DATA_BLOCK "DATA_CONFIG"
{ DB_Accessible_From_OPC_UA := 'FALSE' ;
 S7_Optimized_Access := 'TRUE' }
VERSION : 0.1
NON_RETAIN
   VAR
      PLCVersion { ExternalWritable := 'False'} : String["DIM_STRINGNAME"];   // scritto su Settings
      PLCVersion1 : Int;
      PLCVersion2 : Int;
      PLCVersion3 : Int;
      PLCVersion4 : Int;
      CFGVersion : Int;   // PLCVersion1 * 100 + PLCVersion2
      SerType : Int;   // tipo dati Deserialize
      SerCurrInd : Int;   // indice blocco corrente Deserialize
      SerCurrLast : Int;   // indice ultimo blocco Deserialize
      SerIndStat : Int;
      SerTotRot : Real;
      ConfigReqTime { ExternalAccessible := 'False'; ExternalVisible := 'False'; ExternalWritable := 'False'} : Time;   // NON USATO
      ConfigReqTimeout { ExternalAccessible := 'False'; ExternalVisible := 'False'; ExternalWritable := 'False'} : ULInt;   // NON USATO
      ConfigAckTime { ExternalAccessible := 'False'; ExternalVisible := 'False'; ExternalWritable := 'False'} : Time;   // NON USATO
      ConfigAckTimeout { ExternalAccessible := 'False'; ExternalVisible := 'False'; ExternalWritable := 'False'} : ULInt;   // NON USATO
      ConfigSaveReqTime : Time;
      ConfigSaveReqTimeout : ULInt;
      ConfigSaveReqStart : Bool;
      TabstatReqTime : Time;
      TabstatReqTimeout : ULInt;
      ProgReqHMITime : Time;
      ProgReqHMITimeout : ULInt;
      SaveConfigReq { ExternalAccessible := 'False'; ExternalVisible := 'False'; ExternalWritable := 'False'} : Bool;
      SaveConfigCurrStep { ExternalAccessible := 'False'; ExternalVisible := 'False'; ExternalWritable := 'False'} : Int;
      DeletingFile { ExternalAccessible := 'False'; ExternalVisible := 'False'; ExternalWritable := 'False'} : Bool;
      SavingFile : Bool;   // Scrittura file su WebServer in corso
      DebugInd { ExternalAccessible := 'False'; ExternalVisible := 'False'; ExternalWritable := 'False'} : Int;
      DebugInd2 { ExternalAccessible := 'False'; ExternalVisible := 'False'; ExternalWritable := 'False'} : Int;
      Config_Header { ExternalWritable := 'False'} : Array[0.."MAX_HEADER"] of Int;   // SN,FileType,FileTypeVersion,FileVersion
      AxisFunInd : Array[0.."MAX_ASSEFUNIND"] of Int;
      InInd : Array[0.."MAX_STATOBOOL"] of Int;
      OutInd : Array[0.."MAX_STATOBOOL"] of Int;
      ParamString : Array[0.."MAX_PARAMSTRING"] of String["DIM_STRINGNAME"];
      ParamBool : Array[0.."MAX_PARAMBOOL"] of Bool;
      ParamInt : Array[0.."MAX_PARAMINT"] of Int;
      ParamRealCfg : Array[0.."MAX_PARAMREAL"] of Real;
      ParamReal : Array[0.."MAX_PARAMREAL"] of Real;
      ParamRealType : Array[0.."MAX_PARAMREAL"] of Int;
      ParamRealFC { ExternalAccessible := 'False'; ExternalVisible := 'False'; ExternalWritable := 'False'} : Array[0.."MAX_PARAMREAL"] of Real;
      ParamRealOffset : Array[0.."MAX_PARAMREAL"] of Real;
      IO_Name : Array[0.."MAX_IO"] of String["DIM_STRINGNAME"];
      IO_Param { S7_SetPoint := 'False'} : Array[0.."MAX_IO"] of "Type_IOParam";
      Axis_Name : Array[0.."MAX_ASSE"] of String["DIM_STRINGID"];
      Axis_Param { S7_SetPoint := 'False'} : Array[0.."MAX_ASSE"] of "Type_AxisParam";
      Axis { S7_SetPoint := 'False'} : Array[0.."MAX_ASSE"] of "Type_Axis";
      Input { S7_SetPoint := 'False'} : Array[0.."MAX_INPUT"] of "Type_Input";
      Input_Param { S7_SetPoint := 'False'} : Array[0.."MAX_INPUT"] of "Type_InputParam";
      Feedback { S7_SetPoint := 'False'} : Array[0.."MAX_FEEDBACK"] of "Type_Feedback";
      Feedback_Param { S7_SetPoint := 'False'} : Array[0.."MAX_FEEDBACK"] of "Type_FeedbackParam";
      PID { ExternalAccessible := 'False'; ExternalVisible := 'False'; ExternalWritable := 'False'; S7_SetPoint := 'False'} : Array[0.."MAX_PID"] of "Type_PID";
      PID_Param { S7_SetPoint := 'False'} : Array[0.."MAX_PID"] of "Type_PIDParam";
      Output { S7_SetPoint := 'False'} : Array[0.."MAX_OUTPUT"] of "Type_Output";
      Output_Param { S7_SetPoint := 'False'} : Array[0.."MAX_OUTPUT"] of "Type_OutputParam";
      Motor { S7_SetPoint := 'False'} : Array[0.."MAX_MOTORE"] of "Type_Motor";
      Motor_Config : Array[0.."MAX_MOTORE"] of Bool;
      Motor_Selectable : Array[0.."MAX_MOTORE"] of Bool;
      Motor_LSInd : Array[0.."MAX_MOTORE"] of Int;
      Motor_LS2Ind : Array[0.."MAX_MOTORE"] of Int;
      Motor_CmdInd : Array[0.."MAX_MOTORE"] of Int;
      Motor_Cmd1Ind : Array[0.."MAX_MOTORE"] of Int;
      Motor_Cmd2Ind : Array[0.."MAX_MOTORE"] of Int;
      Motor_Cmd3Ind : Array[0.."MAX_MOTORE"] of Int;
      Motor_StatInd : Array[0.."MAX_MOTORE"] of Int;
      Motor_TRInd : Array[0.."MAX_MOTORE"] of Int;
      Motor_TR2Ind : Array[0.."MAX_MOTORE"] of Int;
      Motor_StartingInd : Array[0.."MAX_MOTORE"] of Int;
      Alarm_Name : Array[0.."MAX_ALARM"] of String["DIM_STRINGNAME"];
      Alarm_Param { S7_SetPoint := 'False'} : Array[0.."MAX_ALARM"] of "Type_AlarmParam";
      Stop_Num : Int;
      Stop_Name : Array[0.."MAX_STOP"] of String["DIM_STRINGNAME"];
      Stop_Ind : Array[0.."MAX_STOP"] of Int;
      Maint_Name : Array[0.."MAX_MAINT"] of String["DIM_STRINGNAME"];
      Maint_Param { S7_SetPoint := 'False'} : Array[0.."MAX_MAINT"] of "Type_MaintParam";
      Toolset_Name { S7_SetPoint := 'True'} : Array[0.."MAX_TOOLSET"] of String["DIM_STRINGNAME"];
      Toolset_Param { S7_SetPoint := 'False'} : Array[0.."MAX_TOOLSET"] of "Type_ToolsetParam";
      UM_FC : Array[0.."MAX_UM"] of Real;
      UM_FC_Met { ExternalAccessible := 'False'; ExternalVisible := 'False'; ExternalWritable := 'False'} : Array[0.."MAX_UM"] of Real;
      UM_FC_Imp { ExternalAccessible := 'False'; ExternalVisible := 'False'; ExternalWritable := 'False'} : Array[0.."MAX_UM"] of Real;
   END_VAR
   VAR RETAIN
      UM_Offset : Array[0.."MAX_UM"] of Real;
   END_VAR
   VAR
      UM_Offset_Met { ExternalAccessible := 'False'; ExternalVisible := 'False'; ExternalWritable := 'False'} : Array[0.."MAX_UM"] of Real;
      UM_Offset_Imp { ExternalAccessible := 'False'; ExternalVisible := 'False'; ExternalWritable := 'False'} : Array[0.."MAX_UM"] of Real;
   END_VAR
   VAR RETAIN
      UM_NDec : Array[0.."MAX_UM"] of Int;
   END_VAR
   VAR
      UM_NDec_Met { ExternalAccessible := 'False'; ExternalVisible := 'False'; ExternalWritable := 'False'} : Array[0.."MAX_UM"] of Int;
      UM_NDec_Imp { ExternalAccessible := 'False'; ExternalVisible := 'False'; ExternalWritable := 'False'} : Array[0.."MAX_UM"] of Int;
   END_VAR
   VAR RETAIN
      UM_Name : Array[0.."MAX_UM"] of String["DIM_STRINGUMNAME"];
   END_VAR
   VAR
      UM_Name_Met { ExternalAccessible := 'False'; ExternalVisible := 'False'; ExternalWritable := 'False'} : Array[0.."MAX_UM"] of String["DIM_STRINGUMNAME"];
      UM_Name_Imp { ExternalAccessible := 'False'; ExternalVisible := 'False'; ExternalWritable := 'False'} : Array[0.."MAX_UM"] of String["DIM_STRINGUMNAME"];
   END_VAR
   VAR RETAIN
      Teach { S7_SetPoint := 'False'} : "Type_Teach";
   END_VAR
   VAR
      Seq { ExternalAccessible := 'False'; ExternalVisible := 'False'; ExternalWritable := 'False'; S7_SetPoint := 'False'} : "Type_Seq";
      HMIAdd0 { ExternalAccessible := 'False'; ExternalVisible := 'False'; ExternalWritable := 'False'} : Int;
   END_VAR


BEGIN
   PLCVersion := '0';
   ConfigReqTime := T#0MS;
   ConfigReqTimeout := 4000;
   ConfigAckTimeout := 4000;
   ConfigSaveReqTimeout := 1500;
   TabstatReqTimeout := 800;
   ProgReqHMITimeout := 1500;
   DebugInd := -1;
   DebugInd2 := -1;
   AxisFunInd[0] := -1;
   AxisFunInd[1] := -1;
   AxisFunInd[2] := -1;
   AxisFunInd[3] := -1;
   AxisFunInd[4] := -1;
   AxisFunInd[5] := -1;
   AxisFunInd[6] := -1;
   AxisFunInd[7] := -1;
   AxisFunInd[8] := -1;
   AxisFunInd[9] := -1;
   AxisFunInd[10] := -1;
   AxisFunInd[11] := -1;
   AxisFunInd[12] := -1;
   AxisFunInd[13] := -1;
   AxisFunInd[14] := -1;
   AxisFunInd[15] := -1;
   AxisFunInd[16] := -1;
   AxisFunInd[17] := -1;
   AxisFunInd[18] := -1;
   AxisFunInd[19] := -1;
   AxisFunInd[20] := -1;
   AxisFunInd[21] := -1;
   AxisFunInd[22] := -1;
   AxisFunInd[23] := -1;
   AxisFunInd[24] := -1;
   AxisFunInd[25] := -1;
   AxisFunInd[26] := -1;
   AxisFunInd[27] := -1;
   AxisFunInd[28] := -1;
   AxisFunInd[29] := -1;
   AxisFunInd[30] := -1;
   AxisFunInd[31] := -1;
   AxisFunInd[32] := -1;
   AxisFunInd[33] := -1;
   AxisFunInd[34] := -1;
   AxisFunInd[35] := -1;
   AxisFunInd[36] := -1;
   AxisFunInd[37] := -1;
   AxisFunInd[38] := -1;
   AxisFunInd[39] := -1;
   AxisFunInd[40] := -1;
   AxisFunInd[41] := -1;
   AxisFunInd[42] := -1;
   AxisFunInd[43] := -1;
   AxisFunInd[44] := -1;
   AxisFunInd[45] := -1;
   AxisFunInd[46] := -1;
   AxisFunInd[47] := -1;
   AxisFunInd[48] := -1;
   AxisFunInd[49] := -1;
   AxisFunInd[50] := -1;
   AxisFunInd[51] := -1;
   AxisFunInd[52] := -1;
   AxisFunInd[53] := -1;
   AxisFunInd[54] := -1;
   AxisFunInd[55] := -1;
   AxisFunInd[56] := -1;
   AxisFunInd[57] := -1;
   AxisFunInd[58] := -1;
   AxisFunInd[59] := -1;
   AxisFunInd[60] := -1;
   AxisFunInd[61] := -1;
   AxisFunInd[62] := -1;
   AxisFunInd[63] := -1;
   AxisFunInd[64] := -1;
   AxisFunInd[65] := -1;
   AxisFunInd[66] := -1;
   AxisFunInd[67] := -1;
   AxisFunInd[68] := -1;
   AxisFunInd[69] := -1;
   AxisFunInd[70] := -1;
   AxisFunInd[71] := -1;
   InInd[0] := -1;
   InInd[1] := -1;
   InInd[2] := -1;
   InInd[3] := -1;
   InInd[4] := -1;
   InInd[5] := -1;
   InInd[6] := -1;
   InInd[7] := -1;
   InInd[8] := -1;
   InInd[9] := -1;
   InInd[10] := -1;
   InInd[11] := -1;
   InInd[12] := -1;
   InInd[13] := -1;
   InInd[14] := -1;
   InInd[15] := -1;
   InInd[16] := -1;
   InInd[17] := -1;
   InInd[18] := -1;
   InInd[19] := -1;
   InInd[20] := -1;
   InInd[21] := -1;
   InInd[22] := -1;
   InInd[23] := -1;
   InInd[24] := -1;
   InInd[25] := -1;
   InInd[26] := -1;
   InInd[27] := -1;
   InInd[28] := -1;
   InInd[29] := -1;
   InInd[30] := -1;
   InInd[31] := -1;
   InInd[32] := -1;
   InInd[33] := -1;
   InInd[34] := -1;
   InInd[35] := -1;
   InInd[36] := -1;
   InInd[37] := -1;
   InInd[38] := -1;
   InInd[39] := -1;
   InInd[40] := -1;
   InInd[41] := -1;
   InInd[42] := -1;
   InInd[43] := -1;
   InInd[44] := -1;
   InInd[45] := -1;
   InInd[46] := -1;
   InInd[47] := -1;
   InInd[48] := -1;
   InInd[49] := -1;
   InInd[50] := -1;
   InInd[51] := -1;
   InInd[52] := -1;
   InInd[53] := -1;
   InInd[54] := -1;
   InInd[55] := -1;
   InInd[56] := -1;
   InInd[57] := -1;
   InInd[58] := -1;
   InInd[59] := -1;
   InInd[60] := -1;
   InInd[61] := -1;
   InInd[62] := -1;
   InInd[63] := -1;
   InInd[64] := -1;
   InInd[65] := -1;
   InInd[66] := -1;
   InInd[67] := -1;
   InInd[68] := -1;
   InInd[69] := -1;
   InInd[70] := -1;
   InInd[71] := -1;
   InInd[72] := -1;
   InInd[73] := -1;
   InInd[74] := -1;
   InInd[75] := -1;
   InInd[76] := -1;
   InInd[77] := -1;
   InInd[78] := -1;
   InInd[79] := -1;
   InInd[80] := -1;
   InInd[81] := -1;
   InInd[82] := -1;
   InInd[83] := -1;
   InInd[84] := -1;
   InInd[85] := -1;
   InInd[86] := -1;
   InInd[87] := -1;
   InInd[88] := -1;
   InInd[89] := -1;
   InInd[90] := -1;
   InInd[91] := -1;
   InInd[92] := -1;
   InInd[93] := -1;
   InInd[94] := -1;
   InInd[95] := -1;
   InInd[96] := -1;
   InInd[97] := -1;
   InInd[98] := -1;
   InInd[99] := -1;
   InInd[100] := -1;
   InInd[101] := -1;
   InInd[102] := -1;
   InInd[103] := -1;
   InInd[104] := -1;
   InInd[105] := -1;
   InInd[106] := -1;
   InInd[107] := -1;
   InInd[108] := -1;
   InInd[109] := -1;
   InInd[110] := -1;
   InInd[111] := -1;
   InInd[112] := -1;
   InInd[113] := -1;
   InInd[114] := -1;
   InInd[115] := -1;
   InInd[116] := -1;
   InInd[117] := -1;
   InInd[118] := -1;
   InInd[119] := -1;
   InInd[120] := -1;
   InInd[121] := -1;
   InInd[122] := -1;
   InInd[123] := -1;
   InInd[124] := -1;
   InInd[125] := -1;
   InInd[126] := -1;
   InInd[127] := -1;
   InInd[128] := -1;
   InInd[129] := -1;
   InInd[130] := -1;
   InInd[131] := -1;
   InInd[132] := -1;
   InInd[133] := -1;
   InInd[134] := -1;
   InInd[135] := -1;
   OutInd[0] := -1;
   OutInd[1] := -1;
   OutInd[2] := -1;
   OutInd[3] := -1;
   OutInd[4] := -1;
   OutInd[5] := -1;
   OutInd[6] := -1;
   OutInd[7] := -1;
   OutInd[8] := -1;
   OutInd[9] := -1;
   OutInd[10] := -1;
   OutInd[11] := -1;
   OutInd[12] := -1;
   OutInd[13] := -1;
   OutInd[14] := -1;
   OutInd[15] := -1;
   OutInd[16] := -1;
   OutInd[17] := -1;
   OutInd[18] := -1;
   OutInd[19] := -1;
   OutInd[20] := -1;
   OutInd[21] := -1;
   OutInd[22] := -1;
   OutInd[23] := -1;
   OutInd[24] := -1;
   OutInd[25] := -1;
   OutInd[26] := -1;
   OutInd[27] := -1;
   OutInd[28] := -1;
   OutInd[29] := -1;
   OutInd[30] := -1;
   OutInd[31] := -1;
   OutInd[32] := -1;
   OutInd[33] := -1;
   OutInd[34] := -1;
   OutInd[35] := -1;
   OutInd[36] := -1;
   OutInd[37] := -1;
   OutInd[38] := -1;
   OutInd[39] := -1;
   OutInd[40] := -1;
   OutInd[41] := -1;
   OutInd[42] := -1;
   OutInd[43] := -1;
   OutInd[44] := -1;
   OutInd[45] := -1;
   OutInd[46] := -1;
   OutInd[47] := -1;
   OutInd[48] := -1;
   OutInd[49] := -1;
   OutInd[50] := -1;
   OutInd[51] := -1;
   OutInd[52] := -1;
   OutInd[53] := -1;
   OutInd[54] := -1;
   OutInd[55] := -1;
   OutInd[56] := -1;
   OutInd[57] := -1;
   OutInd[58] := -1;
   OutInd[59] := -1;
   OutInd[60] := -1;
   OutInd[61] := -1;
   OutInd[62] := -1;
   OutInd[63] := -1;
   OutInd[64] := -1;
   OutInd[65] := -1;
   OutInd[66] := -1;
   OutInd[67] := -1;
   OutInd[68] := -1;
   OutInd[69] := -1;
   OutInd[70] := -1;
   OutInd[71] := -1;
   OutInd[72] := -1;
   OutInd[73] := -1;
   OutInd[74] := -1;
   OutInd[75] := -1;
   OutInd[76] := -1;
   OutInd[77] := -1;
   OutInd[78] := -1;
   OutInd[79] := -1;
   OutInd[80] := -1;
   OutInd[81] := -1;
   OutInd[82] := -1;
   OutInd[83] := -1;
   OutInd[84] := -1;
   OutInd[85] := -1;
   OutInd[86] := -1;
   OutInd[87] := -1;
   OutInd[88] := -1;
   OutInd[89] := -1;
   OutInd[90] := -1;
   OutInd[91] := -1;
   OutInd[92] := -1;
   OutInd[93] := -1;
   OutInd[94] := -1;
   OutInd[95] := -1;
   OutInd[96] := -1;
   OutInd[97] := -1;
   OutInd[98] := -1;
   OutInd[99] := -1;
   OutInd[100] := -1;
   OutInd[101] := -1;
   OutInd[102] := -1;
   OutInd[103] := -1;
   OutInd[104] := -1;
   OutInd[105] := -1;
   OutInd[106] := -1;
   OutInd[107] := -1;
   OutInd[108] := -1;
   OutInd[109] := -1;
   OutInd[110] := -1;
   OutInd[111] := -1;
   OutInd[112] := -1;
   OutInd[113] := -1;
   OutInd[114] := -1;
   OutInd[115] := -1;
   OutInd[116] := -1;
   OutInd[117] := -1;
   OutInd[118] := -1;
   OutInd[119] := -1;
   OutInd[120] := -1;
   OutInd[121] := -1;
   OutInd[122] := -1;
   OutInd[123] := -1;
   OutInd[124] := -1;
   OutInd[125] := -1;
   OutInd[126] := -1;
   OutInd[127] := -1;
   OutInd[128] := -1;
   OutInd[129] := -1;
   OutInd[130] := -1;
   OutInd[131] := -1;
   OutInd[132] := -1;
   OutInd[133] := -1;
   OutInd[134] := -1;
   OutInd[135] := -1;
   ParamRealType[0] := -1;
   ParamRealType[1] := -1;
   ParamRealType[2] := -1;
   ParamRealType[3] := -1;
   ParamRealType[4] := -1;
   ParamRealType[5] := -1;
   ParamRealType[6] := -1;
   ParamRealType[7] := -1;
   ParamRealType[8] := -1;
   ParamRealType[9] := -1;
   ParamRealType[10] := -1;
   ParamRealType[11] := -1;
   ParamRealType[12] := -1;
   ParamRealType[13] := -1;
   ParamRealType[14] := -1;
   ParamRealType[15] := -1;
   ParamRealType[16] := -1;
   ParamRealType[17] := -1;
   ParamRealType[18] := -1;
   ParamRealType[19] := -1;
   ParamRealType[20] := -1;
   ParamRealType[21] := -1;
   ParamRealType[22] := -1;
   ParamRealType[23] := -1;
   ParamRealType[24] := -1;
   ParamRealType[25] := -1;
   ParamRealType[26] := -1;
   ParamRealType[27] := -1;
   ParamRealType[28] := -1;
   ParamRealType[29] := -1;
   ParamRealType[30] := -1;
   ParamRealType[31] := -1;
   ParamRealType[32] := -1;
   ParamRealType[33] := -1;
   ParamRealType[34] := -1;
   ParamRealType[35] := -1;
   ParamRealType[36] := -1;
   ParamRealType[37] := -1;
   ParamRealType[38] := -1;
   ParamRealType[39] := -1;
   ParamRealType[40] := -1;
   ParamRealType[41] := -1;
   ParamRealType[42] := -1;
   ParamRealType[43] := -1;
   ParamRealType[44] := -1;
   ParamRealType[45] := -1;
   ParamRealType[46] := -1;
   ParamRealType[47] := -1;
   ParamRealType[48] := -1;
   ParamRealType[49] := -1;
   ParamRealType[50] := -1;
   ParamRealType[51] := -1;
   ParamRealType[52] := -1;
   ParamRealType[53] := -1;
   ParamRealType[54] := -1;
   ParamRealType[55] := -1;
   ParamRealType[56] := -1;
   ParamRealType[57] := -1;
   ParamRealType[58] := -1;
   ParamRealType[59] := -1;
   ParamRealType[60] := -1;
   ParamRealType[61] := -1;
   ParamRealType[62] := -1;
   ParamRealType[63] := -1;
   ParamRealType[64] := -1;
   ParamRealType[65] := -1;
   ParamRealType[66] := -1;
   ParamRealType[67] := -1;
   ParamRealType[68] := -1;
   ParamRealType[69] := -1;
   ParamRealType[70] := -1;
   ParamRealType[71] := -1;
   ParamRealType[72] := -1;
   ParamRealType[73] := -1;
   ParamRealType[74] := -1;
   ParamRealType[75] := -1;
   ParamRealType[76] := -1;
   ParamRealType[77] := -1;
   ParamRealType[78] := -1;
   ParamRealType[79] := -1;
   ParamRealFC[0] := 1.0;
   ParamRealFC[1] := 1.0;
   ParamRealFC[2] := 1.0;
   ParamRealFC[3] := 1.0;
   ParamRealFC[4] := 1.0;
   ParamRealFC[5] := 1.0;
   ParamRealFC[6] := 1.0;
   ParamRealFC[7] := 1.0;
   ParamRealFC[8] := 1.0;
   ParamRealFC[9] := 1.0;
   ParamRealFC[10] := 1.0;
   ParamRealFC[11] := 1.0;
   ParamRealFC[12] := 1.0;
   ParamRealFC[13] := 1.0;
   ParamRealFC[14] := 1.0;
   ParamRealFC[15] := 1.0;
   ParamRealFC[16] := 1.0;
   ParamRealFC[17] := 1.0;
   ParamRealFC[18] := 1.0;
   ParamRealFC[19] := 1.0;
   ParamRealFC[20] := 1.0;
   ParamRealFC[21] := 1.0;
   ParamRealFC[22] := 1.0;
   ParamRealFC[23] := 1.0;
   ParamRealFC[24] := 1.0;
   ParamRealFC[25] := 1.0;
   ParamRealFC[26] := 1.0;
   ParamRealFC[27] := 1.0;
   ParamRealFC[28] := 1.0;
   ParamRealFC[29] := 1.0;
   ParamRealFC[30] := 1.0;
   ParamRealFC[31] := 1.0;
   ParamRealFC[32] := 1.0;
   ParamRealFC[33] := 1.0;
   ParamRealFC[34] := 1.0;
   ParamRealFC[35] := 1.0;
   ParamRealFC[36] := 1.0;
   ParamRealFC[37] := 1.0;
   ParamRealFC[38] := 1.0;
   ParamRealFC[39] := 1.0;
   ParamRealFC[40] := 1.0;
   ParamRealFC[41] := 1.0;
   ParamRealFC[42] := 1.0;
   ParamRealFC[43] := 1.0;
   ParamRealFC[44] := 1.0;
   ParamRealFC[45] := 1.0;
   ParamRealFC[46] := 1.0;
   ParamRealFC[47] := 1.0;
   ParamRealFC[48] := 1.0;
   ParamRealFC[49] := 1.0;
   ParamRealFC[50] := 1.0;
   ParamRealFC[51] := 1.0;
   ParamRealFC[52] := 1.0;
   ParamRealFC[53] := 1.0;
   ParamRealFC[54] := 1.0;
   ParamRealFC[55] := 1.0;
   ParamRealFC[56] := 1.0;
   ParamRealFC[57] := 1.0;
   ParamRealFC[58] := 1.0;
   ParamRealFC[59] := 1.0;
   ParamRealFC[60] := 1.0;
   ParamRealFC[61] := 1.0;
   ParamRealFC[62] := 1.0;
   ParamRealFC[63] := 1.0;
   ParamRealFC[64] := 1.0;
   ParamRealFC[65] := 1.0;
   ParamRealFC[66] := 1.0;
   ParamRealFC[67] := 1.0;
   ParamRealFC[68] := 1.0;
   ParamRealFC[69] := 1.0;
   ParamRealFC[70] := 1.0;
   ParamRealFC[71] := 1.0;
   ParamRealFC[72] := 1.0;
   ParamRealFC[73] := 1.0;
   ParamRealFC[74] := 1.0;
   ParamRealFC[75] := 1.0;
   ParamRealFC[76] := 1.0;
   ParamRealFC[77] := 1.0;
   ParamRealFC[78] := 1.0;
   ParamRealFC[79] := 1.0;
   Axis_Param[0].realval[51] := 0.0;
   Stop_Ind[0] := -1;
   Stop_Ind[1] := -1;
   Stop_Ind[2] := -1;
   Stop_Ind[3] := -1;
   Stop_Ind[4] := -1;
   Stop_Ind[5] := -1;
   Stop_Ind[6] := -1;
   Stop_Ind[7] := -1;
   Stop_Ind[8] := -1;
   Stop_Ind[9] := -1;
   Stop_Ind[10] := -1;
   Stop_Ind[11] := -1;
   Stop_Ind[12] := -1;
   Stop_Ind[13] := -1;
   Stop_Ind[14] := -1;
   Stop_Ind[15] := -1;
   UM_FC_Met[0] := 1.0;
   UM_FC_Met[1] := 1.0;
   UM_FC_Met[2] := 1.0;
   UM_FC_Met[3] := 1.0;
   UM_FC_Met[4] := 1.0;
   UM_FC_Met[5] := 1.0;
   UM_FC_Met[6] := 1.0;
   UM_FC_Met[7] := 1.0;
   UM_FC_Met[8] := 1.0;
   UM_FC_Met[9] := 1.0;
   UM_FC_Met[10] := 1.0;
   UM_FC_Met[11] := 1.0;
   UM_FC_Met[12] := 1.0;
   UM_FC_Imp[0] := 0.0393701;
   UM_FC_Imp[1] := 14.50377;
   UM_FC_Imp[2] := 1.8;
   UM_FC_Imp[3] := 1.0;
   UM_FC_Imp[4] := 145.0377;
   UM_FC_Imp[5] := 1.0;
   UM_FC_Imp[6] := 0.0393701;
   UM_FC_Imp[7] := 14.50377;
   UM_FC_Imp[8] := 0.001550005;
   UM_FC_Imp[9] := 0.00109361;
   UM_FC_Imp[10] := 145.0377;
   UM_FC_Imp[11] := 1.0;
   UM_FC_Imp[12] := 1.0;
   UM_Offset_Imp[2] := 32.0;
   UM_Offset_Imp[10] := 0.0;
   UM_NDec[9] := 0;
   UM_NDec_Met[0] := 1;
   UM_NDec_Met[2] := 1;
   UM_NDec_Met[6] := 1;
   UM_NDec_Met[7] := 1;
   UM_NDec_Met[9] := 1;
   UM_NDec_Imp[0] := 3;
   UM_NDec_Imp[3] := 1;
   UM_NDec_Imp[4] := 1;
   UM_NDec_Imp[5] := 0;
   UM_NDec_Imp[6] := 2;
   UM_NDec_Imp[7] := 0;
   UM_NDec_Imp[8] := 2;
   UM_NDec_Imp[9] := 1;
   UM_Name[0] := '';
   UM_Name[1] := '';
   UM_Name[2] := '';
   UM_Name[3] := '';
   UM_Name[4] := '';
   UM_Name[5] := '';
   UM_Name[6] := '';
   UM_Name[7] := '';
   UM_Name[8] := '';
   UM_Name[9] := '';
   UM_Name_Met[0] := 'mm';
   UM_Name_Met[1] := 'bar';
   UM_Name_Met[2] := 'C';
   UM_Name_Met[3] := '%';
   UM_Name_Met[4] := 'MPa';
   UM_Name_Met[5] := '%';
   UM_Name_Met[6] := 'mm/sec';
   UM_Name_Met[7] := 'mm/sec2';
   UM_Name_Met[8] := 'mm2';
   UM_Name_Met[9] := 'm';
   UM_Name_Met[10] := 'GPa';
   UM_Name_Met[11] := 'deg';
   UM_Name_Imp[0] := 'in';
   UM_Name_Imp[1] := 'psi';
   UM_Name_Imp[2] := 'F';
   UM_Name_Imp[3] := '%';
   UM_Name_Imp[4] := 'psi';
   UM_Name_Imp[5] := '%';
   UM_Name_Imp[6] := 'in/sec';
   UM_Name_Imp[7] := 'in/sec2';
   UM_Name_Imp[8] := 'in2';
   UM_Name_Imp[9] := 'yd';
   UM_Name_Imp[10] := 'ksi';
   UM_Name_Imp[11] := 'deg';
   Seq.SeqNum := 3;
   Seq.SeqFirst := 0;
   Seq.SeqLast := 2;
   Seq.SeqId[0] := 1;
   Seq.SeqId[1] := 2;
   Seq.SeqId[2] := 3;
   Seq.SeqTyp[0] := 1;
   Seq.SeqTyp[1] := 1;
   Seq.SeqTyp[2] := 1;
   Seq.SeqFirstStat[0] := 0;
   Seq.SeqFirstStat[1] := 2;
   Seq.SeqFirstStat[2] := 3;
   Seq.SeqFirstStat[3] := -1;
   Seq.SeqFirstStat[4] := -1;
   Seq.SeqFirstStat[5] := -1;
   Seq.SeqLastStat[0] := 1;
   Seq.SeqLastStat[1] := 2;
   Seq.SeqLastStat[2] := 3;
   Seq.SeqLastStat[3] := -1;
   Seq.SeqLastStat[4] := -1;
   Seq.SeqLastStat[5] := -1;
   Seq.SeqNext[0] := 1;
   Seq.SeqNext[1] := 2;
   Seq.SeqNext[2] := -1;
   Seq.SeqNext[3] := -1;
   Seq.SeqNext[4] := -1;
   Seq.SeqNext[5] := -1;
   Seq.SeqNumStat[0] := 2;
   Seq.SeqNumStat[1] := 1;
   Seq.SeqNumStat[2] := 1;
   Seq.SeqNumStat[3] := 0;
   Seq.SeqNumStat[4] := 0;
   Seq.SeqNumStat[5] := 0;
   Seq.StatNum := 4;
   Seq.Stat[0].seqid := 1;
   Seq.Stat[0].pos := 0;
   Seq.Stat[0].cod := 0;
   Seq.Stat[0].next := 1;
   Seq.Stat[0].prim := 1;
   Seq.Stat[1].seqid := 1;
   Seq.Stat[1].pos := 1;
   Seq.Stat[1].cod := 3020;
   Seq.Stat[1].prim := 1;
   Seq.Stat[2].seqid := 2;
   Seq.Stat[2].pos := 0;
   Seq.Stat[2].cod := 3215;
   Seq.Stat[2].firstparam := 0;
   Seq.Stat[2].lastparam := 0;
   Seq.Stat[2].next := -1;
   Seq.Stat[2].prim := 1;
   Seq.Stat[3].seqid := 3;
   Seq.Stat[3].pos := 0;
   Seq.Stat[3].cod := 3210;
   Seq.Stat[3].firstparam := 1;
   Seq.Stat[3].lastparam := 1;
   Seq.Stat[3].next := -1;
   Seq.Stat[3].prim := 1;
   Seq.StatParamNum := 2;
   Seq.StatParam[0].seqid := 2;
   Seq.StatParam[0].statpos := 0;
   Seq.StatParam[0].pos := 0;
   Seq.StatParam[0].objtype := 5;
   Seq.StatParam[1].seqid := 3;
   Seq.StatParam[1].statpos := 0;
   Seq.StatParam[1].pos := 0;
   Seq.StatParam[1].objtype := 1;
   Seq.StatParam[1].addr := 31;
   Seq.SeqStartCurrId := -1;
   Seq.SeqStartPrevId := -1;
   Seq.StackLevel := -1;
   Seq.StackLevelAuto := -1;
   Seq.CurrProgSeq := -1;
   Seq.PrevProgSeq := -1;
   HMIAdd0 := 30000;

END_DATA_BLOCK

